TYPE "MatCountCIn"
VERSION : 0.1
// Block: MatCountCIn
   STRUCT
      Rst : Bool;
      Standstill : Bool;
      CheckNextFeeding : Bool;
      EncoderValid : Bool;
      EncoderPosValid : Bool;
      PresetExe : Bool;
      PresetPosition : LReal;
      AxisPos : LReal;
      AxisModule : LReal;
   END_STRUCT;

END_TYPE
